// TIA Portal V18 export
FUNCTION "LGasp_GestioneListaProfila" : Void   // FC10300, LAD
TITLE = Gestione lista profila
{ S7_Optimized_Access := 'TRUE' }
VERSION : 0.1
// stored: AutoNumber true, IsIECCheckEnabled false, SetENOAutomatically false, UDAEnableTagReadback false
   VAR_INPUT
      i_reset_allarmi : Bool;
      i_listaprofila_pezzofatto : "LGasp_typePzoListaProfila";
   END_VAR
   VAR_OUTPUT
      o_listaVuota : Bool;   // lista profila vuota
      o_all_lista_profila_piena : Bool;
   END_VAR
   VAR_IN_OUT
      io_InserisciScartoInListaProfila : Bool;
      io_InserisciPezzoInListaProfila : Bool;
      io_cancella_lista : Bool;
      io_recupero_lista_profila : Bool;
      io_togli_pzo_da_lista : Bool;
      io_lista_pzi : Array[1.."NumMaxPezziProfila"] of "LGasp_typePzoListaProfila";
      io_lista_pzi_backup : Array[1.."NumMaxPezziProfila"] of "LGasp_typePzoListaProfila";
      io_nome_lista_pzi : Array[1.."NumMaxPezziProfila"] of WString[30];   // array letto dal PC
   END_VAR
   VAR_TEMP
      index : Int;
      RigaProduzione_in_lavoro : DInt;
      t_listaVuota : Bool;
      index1 : Int;
      index2 : Int;
   END_VAR
BEGIN

REGION Network 1 (SCL): Descrizione
   //================================================================================
   // Gasparini Spa
   //--------------------------------------------------------------------------------
   // Libreria: LGasp_GestioneListaProfila
   // Funzionalità: Funzione globale per gestione lista profila
   // Commessa in cui è stata testata: 200100305
   // Programmatore di riferimento per test: XXXXXX
   //--------------------------------------------------------------------------------
   // Change log table:
   // Versione     Data           Autore          Modifiche
   //                             M.Dorella       modificata la gestione dello scarto, adesso si possono
   //                                             avere piu'scarti in lista profila non consecutivi
   //              24.01.2022     Lcg             Aggiunta la possibilità di recuperare la lista profila. quando si cancella la lista profila
   //                                             viene fatto un backup. questo è recuperabile se la lista profila è vuota.
   //              01.04.2022      Lcg            Inserimento nome articolo in lista profila (210100012)
   //              06.10.2022      Lcg            Inserita la gestione delle nuove variabili "opzioni" (Bito 210100099) 
   //              29.03.2023      Lcg            Corretto errore che quando si elimina un pezzo da lista profila veniva messo ID a 0 e non -1 (220100026)      
   //-------------------------------------------------------------------------------
   //================================================================================
END_REGION

REGION Network 2 (SCL): inserisci scarto in lista profila
   IF #io_InserisciScartoInListaProfila THEN


       FOR #index1 := 1 TO "NumMaxPezziProfila" - 1 DO//se la lunghezza successiva e' =-1 significa che e' gia' l'ultimo pezzo scarto e non lo inserisco un'altra volta 
           IF #io_lista_pzi[#index1].wastepiece = true AND #io_lista_pzi[#index1 + 1].lenght = -1 THEN
               #io_InserisciScartoInListaProfila := false;
               RETURN;
           END_IF;
       END_FOR;

       FOR #index := 1 TO "NumMaxPezziProfila" DO

                   //inserimento scarto
           IF #io_lista_pzi[#index].lenght = -1.0 THEN
               #io_lista_pzi[#index].ID := 0;
               #io_lista_pzi[#index].name := WSTRING#'';
               #io_lista_pzi[#index].lenght := 0.0;
               #io_lista_pzi[#index].cutoffset := 0.0;
               #io_lista_pzi[#index].NumeroPezzo := 0;
               #io_lista_pzi[#index].wastepiece := true;

               FOR #index2 := 1 TO 16 DO
                   #io_lista_pzi[#index].options[#index2] := FALSE;
               END_FOR;

               #io_lista_pzi[#index].options_dint[1] := -1;
               #io_lista_pzi[#index].options_dint[2] := -1;
               #io_lista_pzi[#index].options_dint[3] := -1;

               #io_lista_pzi[#index].options_lreal[1] := -1.0;
               #io_lista_pzi[#index].options_lreal[2] := -1.0;
               #io_lista_pzi[#index].options_lreal[3] := -1.0;

               #io_lista_pzi[#index].options_str[1] := WSTRING#'';
               #io_lista_pzi[#index].options_str[2] := WSTRING#'';
               #io_lista_pzi[#index].options_str[3] := WSTRING#'';

               EXIT;


           END_IF;

               IF #index = "NumMaxPezziProfila" THEN
                   #o_all_lista_profila_piena := true;
               END_IF;
       END_FOR;
       #io_InserisciScartoInListaProfila := false;
   END_IF;

   IF #i_reset_allarmi THEN
       #o_all_lista_profila_piena := false;
   END_IF;
END_REGION

REGION Network 3 (SCL): inserisci pezzo buono in lista profila
   IF #io_InserisciPezzoInListaProfila THEN
       FOR #index := 1 TO "NumMaxPezziProfila" DO
           IF #io_lista_pzi[#index].lenght = -1.0 THEN
               #io_lista_pzi[#index].ID := #i_listaprofila_pezzofatto.ID;

               //inserimento del nome articolo
               //il nome dell'articolo è appoggiato su un array parallelo alla lista profila perchè in caso di trasferimento ad un altro plc
               //con i-device, un dato wstring non può essere trasferito ma deve essere un array di char.
               //Il pc legge l'array separato dalla lista profila. la linea con le modifiche iniziali è la 210100012
               #io_lista_pzi[#index].name := #i_listaprofila_pezzofatto.name;
               #io_nome_lista_pzi[#index] := #i_listaprofila_pezzofatto.name;

               #io_lista_pzi[#index].lenght := #i_listaprofila_pezzofatto.lenght;
               #io_lista_pzi[#index].cutoffset :=#i_listaprofila_pezzofatto.cutoffset;
               #io_lista_pzi[#index].NumeroPezzo := #i_listaprofila_pezzofatto.NumeroPezzo;
               #io_lista_pzi[#index].wastepiece := false;


               #io_lista_pzi[#index].options := #i_listaprofila_pezzofatto.options;
               #io_lista_pzi[#index].options_dint := #i_listaprofila_pezzofatto.options_dint;
               #io_lista_pzi[#index].options_lreal := #i_listaprofila_pezzofatto.options_lreal;
               #io_lista_pzi[#index].options_str := #i_listaprofila_pezzofatto.options_str;

               EXIT;
           END_IF;

           IF #index = "NumMaxPezziProfila" THEN
               #o_all_lista_profila_piena := true;
           END_IF;
       END_FOR;
       #io_InserisciPezzoInListaProfila := false;
   END_IF;
END_REGION

REGION Network 4 (SCL): svuota lista
   IF #io_cancella_lista = true THEN

       //backup della lista profila per possibile recupero
       IF #io_lista_pzi[1].ID > 0 THEN
           #io_lista_pzi_backup := #io_lista_pzi;
       END_IF;

       #io_cancella_lista := false;

       FOR #index := 1 TO "NumMaxPezziProfila" DO
           #io_lista_pzi[#index].ID := -1;
           #io_lista_pzi[#index].name := WSTRING#'';
           #io_lista_pzi[#index].lenght := -1.0;
           #io_lista_pzi[#index].cutoffset := -1.0;
           #io_lista_pzi[#index].NumeroPezzo := 0;
           #io_lista_pzi[#index].wastepiece := FALSE;

           FOR #index2 := 1 TO 16 DO
               #io_lista_pzi[#index].options[#index2] := FALSE;
           END_FOR;

           #io_lista_pzi[#index].options_dint[1] := -1;
           #io_lista_pzi[#index].options_dint[2] := -1;
           #io_lista_pzi[#index].options_dint[3] := -1;

           #io_lista_pzi[#index].options_lreal[1] := -1.0;
           #io_lista_pzi[#index].options_lreal[2] := -1.0;
           #io_lista_pzi[#index].options_lreal[3] := -1.0;

           #io_lista_pzi[#index].options_str[1] := WSTRING#'';
           #io_lista_pzi[#index].options_str[2] := WSTRING#'';
           #io_lista_pzi[#index].options_str[3] := WSTRING#'';
       END_FOR;
   END_IF;
END_REGION

REGION Network 5 (SCL): Recupero lista profila
   IF #io_recupero_lista_profila THEN

       #io_recupero_lista_profila := false;
       //recupero la lista profila se il backup è valido e la lista è vuota
       IF #io_lista_pzi_backup[1].ID > 0 AND #io_lista_pzi[1].ID = -1 THEN
           #io_lista_pzi := #io_lista_pzi_backup;
       END_IF;

   END_IF;
END_REGION

REGION Network 6 (SCL): togli pezzo da lista profila
   IF #io_togli_pzo_da_lista THEN
       #io_togli_pzo_da_lista := false;

       FOR #index := 1 TO "NumMaxPezziProfila" - 1 DO
           #io_lista_pzi[#index] := #io_lista_pzi[#index + 1];
           IF #io_lista_pzi[#index + 1].lenght = -1.0 THEN
               EXIT;
           END_IF;
       END_FOR;

       #io_lista_pzi[NumMaxPezziProfila].ID := -1;
       #io_lista_pzi[#index].name := WSTRING#'';
       #io_lista_pzi[NumMaxPezziProfila].lenght := -1.0;
       #io_lista_pzi[NumMaxPezziProfila].cutoffset := -1.0;
       #io_lista_pzi[NumMaxPezziProfila].NumeroPezzo := 0;
       #io_lista_pzi[NumMaxPezziProfila].wastepiece := FALSE;

       FOR #index2 := 1 TO 16 DO
           #io_lista_pzi[NumMaxPezziProfila].options[#index2] := FALSE;
       END_FOR;
       #io_lista_pzi[NumMaxPezziProfila].options_dint[1] := -1;
       #io_lista_pzi[NumMaxPezziProfila].options_dint[2] := -1;
       #io_lista_pzi[NumMaxPezziProfila].options_dint[3] := -1;

       #io_lista_pzi[NumMaxPezziProfila].options_lreal[1] := -1.0;
       #io_lista_pzi[NumMaxPezziProfila].options_lreal[2] := -1.0;
       #io_lista_pzi[NumMaxPezziProfila].options_lreal[3] := -1.0;

       #io_lista_pzi[NumMaxPezziProfila].options_str[1] := WSTRING#'';
       #io_lista_pzi[NumMaxPezziProfila].options_str[2] := WSTRING#'';
       #io_lista_pzi[NumMaxPezziProfila].options_str[3] := WSTRING#'';
   END_IF;
END_REGION

REGION Network 7 (SCL): Info lista vuota
   #t_listaVuota := TRUE;
   FOR #index := 1 TO "NumMaxPezziProfila" DO
       IF 0 <> #io_lista_pzi[#index].ID THEN
           #t_listaVuota := FALSE;
           EXIT;
       END_IF;
   END_FOR;
   #o_listaVuota := #t_listaVuota;
END_REGION
END_FUNCTION
